PROGRAM MAIN
VAR
	a10	: BOOL;
END_VAR

END_PROGRAM

(* stored: Version 1.1.0.1
   POU MAIN: Id {9b544d30-5de0-4bac-a48a-e1f991a5356f} *)
